FUNCTION_BLOCK FT_PT2 (* 2nd grade filter with programmable times *)
  (* Standard: 61499-1 *)
  (* Version 1.5, 2025-12-21, franz *)
  PACKAGE OSCAT::Basic::POUs::Engineering::Control;
  IMPORT OSCAT::Basic::POUs::conversion::TIME_TO_REAL;
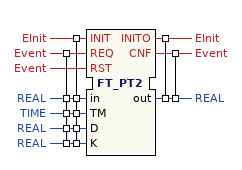
  EVENT_INPUT
    INIT : EInit WITH in, TM, D, K; (* Init Request *)
    REQ WITH in, TM, D, K; (* Normal Execution Request *)
    RST; (* Reset Filter *)
  END_EVENT
  EVENT_OUTPUT
    INITO : EInit WITH out; (* Init Confirmation *)
    CNF WITH out; (* Execution Confirmation *)
  END_EVENT
  VAR_INPUT
    in : REAL; (* Input Signal *)
    TM : TIME; (* Time Constant *)
    D : REAL; (* Damping Factor *)
    K : REAL := 1.0; (* Gain *)
  END_VAR
  VAR_OUTPUT
    out : REAL; (* Filtered Output *)
  END_VAR
  VAR
    init : BOOL := FALSE;
    TN : REAL;
    I1 : REAL;
    I2 : REAL;
    tn2 : REAL;
  END_VAR
  FBS
    int1 : OSCAT::Basic::POUs::Engineering::Control::INTEGRATE;
    int2 : OSCAT::Basic::POUs::Engineering::Control::INTEGRATE;
  END_FBS
  EC_STATES
    INIT : INIT -> INITO;
    REQ : REQ -> CNF;
    RST : RST -> CNF;
  END_STATES
  ALGORITHM INIT IN ST:
(* Startup Initialization *)
init := FALSE;
  END_ALGORITHM
  ALGORITHM RST IN ST:
init := TRUE;
out := K * in;
I2 := out;
  END_ALGORITHM
  ALGORITHM REQ IN ST:
ALGORITHM REQ
(* startup initialisation *)
IF NOT init OR TM = T#0s THEN
	this.RST();
ELSE
	TN := TIME_TO_REAL(TM) * 1.0E-3;
	tn2 := TN * TN;
	int1.REQ(X := in * K / tn2 - I1 * 0.5 * D / TN - I2 / tn2, Y := I1);
	int2.REQ(X := I1, Y := I2);
	out := I2;
END_IF;
END_ALGORITHM

(* revision history
 * *
 * 15.1.2007 hm		rev 1.1 changed formula to new more acurate formula
 * *
 * hm 15.9.2007		rev 1.2 deleted unused code for init system time reading tx
 * *
 * hm	30.11.2007	rev 1.3 changed out to be K * in during initialization avoind divide by 0 if tn
 * = 0
 * *
 * hm	3. nov. 2008	rev 1.4 optimized code and fixed a problem with init
 * *
 * hm	11. mar. 2009	rev 1.5 real constants updated to new systax using dot
 * * *)
  END_ALGORITHM
END_FUNCTION_BLOCK
